FUNCTION_BLOCK PWM
VAR_INPUT
	bVar: BOOL;
		tTime: LTIME;

END_VAR
VAR_OUTPUT
		Led1: BOOL;
END_VAR
VAR
	nState: INT;
	LTON1: LTON;
	LTON2: LTON;
	toplamT: LTIME;
	realVal1: LREAL;
	realVal2: LREAL;
	newTime: LTIME;
END_VAR

toplamT:=LTIME#200US;
realVal1:=LTIME_TO_LREAL(tTime);
realVal2:=LTIME_TO_LREAL(toplamT);

newTime:=LREAL_TO_LTIME(realVal2-realVal1);

CASE nState OF
	
0:
	IF bVar THEN
	
		nState:=10;
	
	END_IF

10:
	
	Led1:=TRUE;
	LTON1(IN:=TRUE , PT:=tTime , Q=> , ET=> );
	
	IF Lton1.Q THEN

		nState:=20;	
		LTON1(IN:=FALSE);
		
	END_IF

20:
	
	Led1:=FALSE;
	LTON2(IN:=TRUE , PT:=newTime , Q=> , ET=> );
	
	IF Lton2.Q THEN

		nState:=0;	
		LTON2(IN:=FALSE);
		
	END_IF
END_CASE

	IF NOT(bVar) THEN

		nState:=0;	
		LTON2(IN:=FALSE);
		LTON1(IN:=FALSE);

	END_IF

END_FUNCTION_BLOCK

(* stored: Version 1.1.0.1, ProductVersion 3.1.4024.4
   POU PWM: Id {6e07600c-f476-4ae1-8f9c-980c015ead37}, SpecialFunc None *)
